# B&R Automation Studio project AriesV2 (part 4)

### Generic_Controls.typ - Global data types
```iecst
(********************************************************************
 * COPYRIGHT --
 ********************************************************************
 * Package: HMI_Visu
 * File: HMI_Visu.typ
 * Author: John
 * Created: February 03, 2015
 ********************************************************************
 * Data types of package HMI_Visu
 ********************************************************************)

TYPE
	Generic_HMI_Ctrl : 	STRUCT
		Ctrl : HMI_Ctrl_typ;
		Data : HMI_Data_typ;
END_STRUCT;
	HMI_Ctrl_typ : 	STRUCT
		KeyLevel : HMI_Control_Change_Current;
		Language : HMI_Control_Change_Current;
		Page : HMI_Control_Change_Current;
		Screensaver : HMI_Control_ScreenTimer;
		Backlight : HMI_Control_ScreenTimer;
		Calibration : HMI_Control_Calibration;
END_STRUCT;
	HMI_Control_Calibration : 	STRUCT
		State : USINT;
		DataPoint : USINT;
END_STRUCT;
	HMI_Control_ScreenTimer : 	STRUCT
		Time_Remaining : UDINT;
		Time_Until_Display : UDINT;
END_STRUCT;
	HMI_Data_typ : 	STRUCT
		Wheel : HMI_Data_Wheel_typ;
END_STRUCT;
	HMI_Data_Wheel_typ : 	STRUCT
		Enter : BOOL;
		Counts : DINT;
END_STRUCT;
	HMI_Control_Change_Current : 	STRUCT
		Change : DINT;
		Current : DINT;
END_STRUCT;
	Listbox_Option_Enum :
		(
		ALLOW := 0,
		DISALLOW := 1,
		HIDDEN := 2
);
	GenericListbox_typ : 	STRUCT
		Strings : ARRAY[0..Enum_Max_Listbox_Items]OF STRING[Enum_Max_Listbox_Char];
		Index : DINT;
		maxidx : USINT;
		minidx : USINT;
		status : USINT;
		option : ARRAY[0..Enum_Max_Listbox_Items]OF USINT;
END_STRUCT;
	GenericButton_typ : 	STRUCT
		datapoint : USINT;
		status : USINT;
		text : STRING[64];
END_STRUCT;
END_TYPE
```

### Program Logical/HMI/hmilogic (ANSIC) - Service that manages navigating through the VC4 HMI

#### loginCyclicLogic.c
```c
#include <bur/plctypes.h>
#ifdef _DEFAULT_INCLUDES
#include <AsDefault.h>
#endif

void loginLevelParameterEditControl(UDINT minLevel)
{
	//input form (i.e. common page) not visible for operator
	//(i.e. loginlevel==0 > visibility set to 1 (not visible))
	gHmiParamTable.selValueFormVisible = (gHmi.prv.loginLevel >= minLevel) ? 0 : 1;
}

//login level related logic
void	loginLevelLogicCyclic()
{
	static UINT loginLevelOld;

	//update visiblity flags that are associated with the current login level
	//note that current app support three login levels: 0-operator;1-supervisor;2-admin
	if(gHmi.prv.loginLevel == 1){
		gHmi.status.loginVisibleGE1 = 0;//visible
		gHmi.status.loginVisibleGE2 = 1;//not visible
		gHmi.status.loginVisibleGE3 = 1;//not visible
	}else
		if(gHmi.prv.loginLevel == 2){
		gHmi.status.loginVisibleGE1 = 0;//visible
		gHmi.status.loginVisibleGE2 = 0;//visible
		gHmi.status.loginVisibleGE3 = 1;//not visible
	}else
		if(gHmi.prv.loginLevel == 3){
		gHmi.status.loginVisibleGE1 = 0;//visible
		gHmi.status.loginVisibleGE2 = 0;//visible
		gHmi.status.loginVisibleGE3 = 0;//visible
	}else{
		gHmi.status.loginVisibleGE1 = 1;//not visible
		gHmi.status.loginVisibleGE2 = 1;//not visible
		gHmi.status.loginVisibleGE3 = 1;//not visible
	}

	//operate login timeout timer
	//Timer for timed out operation of the access control

	bgTimerCyclic(&gHmi.prv.tmr3) ;

	//detect login level changes
	if(gHmi.prv.loginLevel != loginLevelOld){
		loginLevelOld = gHmi.prv.loginLevel;
		if(gHmi.prv.loginLevel){
			//when supervisor or admin logs in > start login timeout timer
			bgTimerStart(&gHmi.prv.tmr3, Tms(DEFINE_LOGIN_TO)); //login duration timer setting comes from current config [sec], convert to [ms]
		}else{
			//when loginLevel gets reset to 0, make sure to make the parametar input field invisible
			loginLevelParameterEditControl(1);
		}
	}

	//restart login timer if user touches the area of the ticking logout timer
	if(gHmi.keys.btnRestartLoginTimer){
		gHmi.keys.btnRestartLoginTimer = 0;
		bgTimerStart(&gHmi.prv.tmr3, Tms(DEFINE_LOGIN_TO));
	}

	//change page to login is user touches the area of the login icon
	if(gHmi.keys.btnLoginIcon){
		gHmi.keys.btnLoginIcon = 0;
		if(!gHmi.prv.loginLevel){
			gHmi.prv.changePage = HMI_LOGIN_40_MAIN;
		}
	}

	//timer based logout > if loginLeve higher then 0, reset it after timer expires
	if(gHmi.prv.loginLevel && bgTimerIsTimeOut(&gHmi.prv.tmr3)){
		gHmi.prv.loginLevel = 0;
	}

	//calculate remaining login time [min:sec] from remaining timer time [ms]
	gHmi.prv.tmr3RemainingTimeSec = (bgTimerTimeRemaining(&gHmi.prv.tmr3)/1000) % 60;
	gHmi.prv.tmr3RemainingTimeMin = (bgTimerTimeRemaining(&gHmi.prv.tmr3)/1000) / 60;

}
```

### Program Logical/HMI/ForceIO (IEC)

#### Variables.var
```iecst
VAR
	pToggle : REFERENCE TO BOOL;
	pSet : REFERENCE TO BOOL;
	pReset : REFERENCE TO BOOL;
	pForceIOPt : REFERENCE TO BOOL;
	ii_force : UDINT := 0;
END_VAR
```

#### Main.st
```iecst
PROGRAM _INIT
//	gHMIForceIO.forceItems[0].pAddrIO := ADR(ControlIO.iRunCmd);
//	gHMIForceIO.forceItems[1].pAddrIO := ADR(ControlIO.iReservoirLevel);
//	gHMIForceIO.forceItems[2].pAddrIO := ADR(CureIO.oUVCureChannel[0]);
//	gHMIForceIO.forceItems[3].pAddrIO := ADR(CureIO.oUVCureChannel[1]);
//	gHMIForceIO.forceItems[4].pAddrIO := ADR(StatusIO.iClearError);
//	gHMIForceIO.forceItems[5].pAddrIO := ADR(ControlIO.iTargetPiP);
//	gHMIForceIO.forceItems[6].pAddrIO := ADR(ControlIO.oTargetPresent);
//	gHMIForceIO.forceItems[7].pAddrIO := ADR(StatusIO.oRunningReady);
END_PROGRAM

PROGRAM _CYCLIC
	IF gHMIForceIO.forceEnable = 0 THEN //IMPORTANTTODO: only go to max idx! FIX THIS IN AS5200 AND UVF AS WELL!
		gHMIForceIO.forceItemsVisibility := 1;

		FOR ii_force := 0 TO HMI_ENUM_FORCEIO_LASTINDEX BY 1 DO
			pForceIOPt ACCESS gHMIForceIO.forceItems[ii_force].pAddrIO;
			pSet ACCESS ADR(gHMIForceIO.forceItems[ii_force].set);
			pReset ACCESS ADR(gHMIForceIO.forceItems[ii_force].reset);
			pToggle ACCESS ADR(gHMIForceIO.forceItems[ii_force].toggle);

			pSet := FALSE;
			pReset := FALSE;
			pToggle := FALSE;
		END_FOR;
	ELSE
		gHMIForceIO.forceItemsVisibility := 0;

		FOR ii_force := 0 TO HMI_ENUM_FORCEIO_LASTINDEX BY 1 DO
			IF gHMIForceIO.forceItems[ii_force].pAddrIO <> 0 THEN
				pForceIOPt ACCESS gHMIForceIO.forceItems[ii_force].pAddrIO;
				pSet ACCESS ADR(gHMIForceIO.forceItems[ii_force].set);
				pReset ACCESS ADR(gHMIForceIO.forceItems[ii_force].reset);
				pToggle ACCESS ADR(gHMIForceIO.forceItems[ii_force].toggle);

				IF pSet THEN
					pForceIOPt := TRUE;
				END_IF;

				IF pReset THEN
					pForceIOPt := FALSE;
				END_IF;

				IF pToggle THEN
					pToggle := FALSE;
					pForceIOPt := NOT pForceIOPt;
				END_IF;
			END_IF;
		END_FOR;
	END_IF;

END_PROGRAM

PROGRAM _EXIT
	(* Insert code here *)

END_PROGRAM
```

### Program Logical/HMI/HMITableManager (IEC) - Manage activating the PV List tables for recipe, configuration params (gRecCfg.active.<>)

#### Main.st
```iecst
//     __ __                         __  ___               ___         __           _             ____
//    / // /__ _______  ___  ___    /  |/  /__ ____  __ __/ _/__ _____/ /___ ______(_)__  ___ _  /  _/__  ____
//   / _  / -_) __/ _ \/ _ \/ _ \  / /|_/ / _ `/ _ \/ // / _/ _ `/ __/ __/ // / __/ / _ \/ _ `/ _/ // _ \/ __/
//  /_//_/\__/_/ /_//_/\___/_//_/ /_/  /_/\_,_/_//_/\_,_/_/ \_,_/\__/\__/\_,_/_/ /_/_//_/\_, / /___/_//_/\__(_)
//                                                                                      /___/
//  Copyright
PROGRAM _INIT
	Init_Logbook.Enable := TRUE;
	Init_Logbook.Name := 'usr_table';
	Init_Logbook();

	//loadHMITable is a FBK with structures containing the values loaded from the textsystem files
	loadHMITable[TABLE_REC_CONTROL]		(tableName := 'Control Recipe',				nameSpace := 'hmiTable/Rec/Control',		Logbook := Init_Logbook.pLog, 	pOverallStats := ADR(tableStats.Overall));
	loadHMITable[TABLE_REC_DISPENSE]	(tableName := 'Dispense Recipe',			nameSpace := 'hmiTable/Rec/Dispense',		Logbook := Init_Logbook.pLog, 	pOverallStats := ADR(tableStats.Overall));
	loadHMITable[TABLE_CFG_CONTROL]		(tableName := 'Control Configuration',		nameSpace := 'hmiTable/Cfg/Control',		Logbook := Init_Logbook.pLog, 	pOverallStats := ADR(tableStats.Overall));
	loadHMITable[TABLE_CFG_DISPENSE]	(tableName := 'Dispense Configuration',		nameSpace := 'hmiTable/Cfg/Dispense',		Logbook := Init_Logbook.pLog, 	pOverallStats := ADR(tableStats.Overall));
END_PROGRAM

//TODO: Load param array with %s, replace with index.
//TODO: More scrutiny to ensure tables were done correctly

PROGRAM _CYCLIC
	IF gHmi.tables.Trigger.Rec.Control THEN
		gHmi.tables.Trigger.Rec.Control := FALSE;
		ActivateHMITable(gRecCfg.active.Cfg.HMI.MachineLang, pHMITable := ADR(gHmiParamTable), pTableValues := ADR(loadHMITable[TABLE_REC_CONTROL].hmiStruct));//No Control recipe values
	END_IF;

	IF gHmi.tables.Trigger.Rec.Dispense THEN
		gHmi.tables.Trigger.Rec.Dispense := FALSE;
		ActivateHMITable(gRecCfg.active.Cfg.HMI.MachineLang, pHMITable := ADR(gHmiParamTable), pTableValues := ADR(loadHMITable[TABLE_REC_DISPENSE].hmiStruct));
	END_IF;

	IF gHmi.tables.Trigger.Cfg.Control THEN
		gHmi.tables.Trigger.Cfg.Control := FALSE;
		ActivateHMITable(gRecCfg.active.Cfg.HMI.MachineLang, pHMITable := ADR(gHmiParamTable), pTableValues := ADR(loadHMITable[TABLE_CFG_CONTROL].hmiStruct));
	END_IF;

	IF gHmi.tables.Trigger.Cfg.Dispense THEN
		gHmi.tables.Trigger.Cfg.Dispense := FALSE;
		ActivateHMITable(gRecCfg.active.Cfg.HMI.MachineLang, pHMITable := ADR(gHmiParamTable), pTableValues := ADR(loadHMITable[TABLE_CFG_DISPENSE].hmiStruct));
	END_IF;

	IF gHmi.tables.Load.Trigger THEN
		SYSreset(1,1);
	END_IF;

	hmiParamListTableCyclic(ADR(gHmiParamTable));

END_PROGRAM
```

- Visualisation Logical/HMI/Visu (not shown)

### Package Logical/Axisobj - Axisobj

### Axisi.ax
```
InitParameter (Version=3.16.1, NcSwId=ACP10)
  ACP10AXIS_typ:
    dig_in:
      level:
        reference = ncACTIV_HI
        pos_hw_end = ncACTIV_HI
        neg_hw_end = ncACTIV_HI
        trigger1 = ncACTIV_HI
        trigger2 = ncACTIV_HI
    encoder_if:
      parameter:
        count_dir = ncSTANDARD
        scaling:
          load:
            units = 125664
            rev_motor = 5
    limit:
      parameter:
        v_pos = 1.0E+08
        v_neg = 1.0E+08
        a1_pos = 1.0E+08
        a2_pos = 1.0E+08
        a1_neg = 1.0E+08
        a2_neg = 1.0E+08
        t_jolt = 0.0
        t_in_pos = 0.1
        pos_sw_end = 2147483647
        neg_sw_end = -2147483648
        ds_warning = 1000.0
        ds_stop = 1000.0
        a_stop = 1.0E+30
        dv_stop = 0.0
        dv_stop_mode = ncOFF
    controller:
      mode = ncPOSITION
      position:
        kv = 50.0
        tn = 0.0
        t_predict = 0.0004
        t_total = 0.0004
        p_max = 1.0E+30
        i_max = 1.0E+30
      speed:
        kv = 1.7
        tn = 1.0
        t_filter = 0.0
        isq_filter1:
          type = ncOFF
          a0 = 0.0
          a1 = 0.0
          b0 = 0.0
          b1 = 0.0
          b2 = 0.0
          c0_par_id = 0
          c1_par_id = 0
        isq_filter2:
          type = ncOFF
          a0 = 0.0
          a1 = 0.0
          b0 = 0.0
          b1 = 0.0
          b2 = 0.0
          c0_par_id = 0
          c1_par_id = 0
        isq_filter3:
          type = ncOFF
          a0 = 0.0
          a1 = 0.0
          b0 = 0.0
          b1 = 0.0
          b2 = 0.0
          c0_par_id = 0
          c1_par_id = 0
      uf:
        type = ncLINEAR
        auto_config = ncMOTOR_PAR
        u0 = 0.0
        un = 0.0
        fn = 50.0
        k_f_slip = 0.0
      ff:
        torque_load = 0.0
        torque_pos = 0.0
        torque_neg = 0.0
        kv_torque = 0.0
        inertia = 0.0
        t_filter_a = 0.0
    move:
      stop:
        parameter[0]:
          decel_ramp = ncA_LIMIT
          controller = ncON
        parameter[1]:
          decel_ramp = ncA_LIMIT
          controller = ncON
        parameter[2]:
          decel_ramp = ncA_LIMIT
          controller = ncON
        parameter[3]:
          decel_ramp = ncA_LIMIT
          controller = ncON
        quickstop:
          decel_ramp = ncA_LIMIT
        drive_error:
          decel_ramp = ncA_LIMIT
      homing:
        parameter:
          s = 0
          v_switch = 5000.0
          v_trigger = 500.0
          a = 50000.0
          mode = ncDIRECT
          edge_sw = ncPOSITIVE
          start_dir = ncPOSITIVE
          trigg_dir = ncPOSITIVE
          ref_pulse = ncOFF
          fix_dir = ncOFF
          tr_s_block = 0.0
          torque_lim = 0.0
          ds_block = 0.0
          ds_stop = 0.0
      basis:
        parameter:
          v_pos = 100000.0
          v_neg = 100000.0
          a1_pos = 200000.0
          a2_pos = 200000.0
          a1_neg = 200000.0
          a2_neg = 200000.0
    message:
      text:
        parameter:
          format = ncBREAK + ncZERO
          columns = 80
          data_modul = acp10etxen
```

### GlobalConstants.var - not listed in the package file held
```iecst
VAR CONSTANT
	FORCEIO_ACCESS_LEVEL : UINT := 1;
	CONFIG_ACCESS_LEVEL : UINT := 2;
	RECIPE_ACCESS_LEVEL : UINT := 1;
	DEFINE_MENU_L_HIDE_TIMEOUT_MS : UDINT := 7000;
	DEFINE_MENU_R_HIDE_TIMEOUT_MS : UDINT := 7000;
	DEFINE_HMI_SPLASHSCREEN_TO_MS : UDINT := 5000;
	MAX_IDX_TOTAL_RECIPES : UINT := 100;
	DEFINE_LOGIN_TO : REAL := 600; (*// at timer DEFINE_LOGIN_TO * 1000 *60*)
END_VAR
(*Insert your comment here.*)
VAR CONSTANT
	MAX_IDX_CREASES : UDINT := 9;
END_VAR
(*Insert your comment here.*)
(*Insert your comment here.*)
VAR RETAIN
	gRecCfg : Global_Par_typ;
END_VAR
VAR
	gAlarms : Machine_Alarms_typ;
	gMachineName : {REDUND_UNREPLICABLE} STRING[80] := 'AS3500HS';
	gProjectDate : {REDUND_UNREPLICABLE} STRING[80] := '7. March 2017';
	gVersion : {REDUND_UNREPLICABLE} STRING[80] := 'TBD';
END_VAR
(*Insert your comment here.*)
VAR
	Axis1 : ACP10AXIS_typ;
	AxisControl : MpAxisBasic;
	AxisPar : MpAxisBasicParType;
END_VAR
(*Insert your comment here.*)
VAR
	MachineState : AriesMachineState_Enum;
	ProcessState : CreaserPrcsState_Enum;
END_VAR
(*Insert your comment here.*)
VAR
	IO : AriesIOPoints_typ;
	IO_LastCycle : AriesIOPoints_typ;
END_VAR
(*Insert your comment here.*)
VAR RETAIN
	gStatistics : Global_Statistics_typ;
END_VAR
(*Insert your comment here.*)
(*Insert your comment here.*)
(*Insert your comment here.*)
(*Insert your comment here.*)
```

### Program Logical/MotionControl/LineControl

#### Variables.var
```iecst
VAR
	pAxisControl : REFERENCE TO MpAxisBasic;
	pAxisPar : REFERENCE TO MpAxisBasicParType;
END_VAR
```

#### Main.st
```iecst
PROGRAM _INIT

END_PROGRAM

PROGRAM _CYCLIC

	pAxisControl ACCESS ADR(AxisControl);
	pAxisPar ACCESS ADR(AxisPar);

END_PROGRAM

PROGRAM _EXIT
	(* Insert code here *)

END_PROGRAM
```

Listed in the project but not available here: Logical/Libraries/MAPPSuppor/MAPPSuppor.typ, Logical/Libraries/MAPPSuppor/HMIparamList.typ, Logical/Libraries/MAPPSuppor/MAPPSuppor.var, Logical/Libraries/MAPPSuppor/MAPPSuppor.fun, Logical/Libraries/MAPPSuppor/hmiParamList.h, Logical/Libraries/MAPPSuppor/hmiParamList.c, Logical/Libraries/MAPPSuppor/bgstring.c, Logical/Libraries/MAPPSuppor/bgstring.h, Logical/Libraries/MAPPSuppor/bgsprintf.c, Logical/Libraries/MAPPSuppor/FBK_Init_Logbook.c, Logical/Libraries/MAPPSuppor/hmiTableFBK_typ.c, Logical/Libraries/wbrServices/Cyclic/wbrService/wbrServiceCyclic.c, Logical/Libraries/wbrServices/wbrListSvc/wbrListSvc.typ, Logical/Libraries/wbrServices/wbrListSvc/wbrListSvc.var, Logical/Libraries/wbrServices/wbrListSvc/wbrListSvc.fun, Logical/Libraries/wbrServices/wbrListSvc/wbrListSvc.c, Logical/Application/Creaser/Types.typ, Logical/Application/Creaser/Action_Stop_Feeder.st, Logical/Application/Creaser/Action_Move_Crease_Width.st, Logical/Application/Creaser/LocalFunctions.fun, Logical/Application/Creaser/PulseTrain.st, Logical/Application/Creaser/Action_Move_Photoeye_Offset.st, Logical/Application/Creaser/Action_Init_Infeed_Axis.st, Logical/Application/Creaser/Action_CreaserProcess_SM.st, Logical/Application/Dispense/Valves, Logical/HMI/HMI_Pages.typ, Logical/HMI/HMIdialog.typ, Logical/HMI/HMImsgScroll.typ, Logical/HMI/HMIForceIO.typ, Logical/HMI/HMIalert.typ, Logical/HMI/HMI.typ, Logical/HMI/HMIremmem.typ, Logical/HMI/HMI.var, Logical/HMI/hmilogic/hmilogic.c, Logical/HMI/hmilogic/hmiParamList.c, Logical/HMI/hmilogic/hmiDialog.c, Logical/HMI/hmilogic/hmiAlert.c, Logical/HMI/hmilogic/loginLogic_Header.h, Logical/HMI/hmilogic/hmiParamList.h, Logical/HMI/hmilogic/hmiAlert.h, Logical/HMI/hmilogic/hmiDialog.h, Logical/HMI/hmilogic/HMIlocal.var, Logical/HMI/HMI_Alarms, Logical/acp10etxen
